// TIA Portal V20 export
// export: Created 2026-07-10T11:12:32.3020878Z, ExportSetting WithDefaults, DisplayName Totally Integrated Automation Portal, DisplayVersion V20, DisplayName TIA Portal Openness, DisplayVersion V20, DisplayName TIA Portal Version Control Interface, DisplayVersion V20, DisplayName STEP 7 Professional, DisplayVersion V20, DisplayName STEP 7 Safety, DisplayVersion V20, DisplayName WinCC Basic/Comfort/Advanced, DisplayVersion V20, DisplayName WinCC Unified, DisplayVersion V20
FUNCTION_BLOCK "PIDRegulator"   // FB9, SCL
{ S7_Optimized_Access := 'TRUE' }
VERSION : 0.1
// stored: AutoNumber true, IsIECCheckEnabled false, IsRetainMemResEnabled false, MemoryReserve 100, SetENOAutomatically false, UDAEnableTagReadback false
   VAR_INPUT
      Enable : Bool;
      Tanklevel : Real;
      TankLevelSetpoint : Real;
      KP : Real := 2.0;
      KI : Real := 0.2;
      KD : Real := 0.5;
      TI : Time := T#1s;
      LimitMin : Real := -100.0;
      LimitMax : Real := 100.0;
      DeadZone : Real := 1.0;
   END_VAR
   VAR_OUTPUT
      DamperPosition : Real;
   END_VAR
   VAR
      "e" : Real;
      PValue : Real;
      IValue : Real;
      DValue : Real;
      init : Bool;
      TopLevelSetPoint : Real;
      BottomlevelSetPoint : Real;
      PrevValue : Real;
      TON1 { S7_SetPoint := 'True'} : TON_TIME;
   END_VAR
BEGIN
   IF NOT #Enable THEN
       #init := false;
       #IValue := 0;
       #DValue := 0;
   END_IF;

   IF NOT #init THEN
       #PrevValue := #Tanklevel;
       #init := TRUE;
   END_IF;

   #TopLevelSetPoint := #TankLevelSetpoint + #DeadZone;
   #BottomlevelSetPoint := #TankLevelSetpoint - #DeadZone;

   IF #Tanklevel > #TopLevelSetPoint THEN
       #e := #TopLevelSetPoint - #Tanklevel;
   ELSIF #Tanklevel < #BottomlevelSetPoint THEN
       #e := #BottomlevelSetPoint - #Tanklevel;
   ELSE
       #e := 0;
       #PrevValue := #Tanklevel;
   END_IF;



   #TON1(IN:=TRUE,
         PT:=#TI);



   IF #TON1.Q THEN
       #IValue := #IValue + #e * #KI;
       #IValue := LIMIT(MN := #LimitMin, IN := #IValue, MX := #LimitMax);

       IF #KI <= 0.00001 THEN
           #IValue := 0;
       END_IF;
       #PValue := #e * #KP;
       #DValue := (#Tanklevel - #PrevValue) * #KD;
       #PrevValue := #Tanklevel;
       #DamperPosition := #PValue + #IValue - #DValue;
       RESET_TIMER(#TON1);
   END_IF;
END_FUNCTION_BLOCK
